% RSLogix 500 project I2P-JOB-15 Duncan_Sutton.RSS, saved by version 10.00.00.00 %
PROJECT "ML01A"    % processor: Bul.1763 MicroLogix 1100 Series B %

PROGRAM FILES
  LAD 2   15 rungs

DATA FILES
  O0 OUTPUT  4 elements
  I1 INPUT  6 elements
  S2 STATUS  66 elements
  B3 BINARY  1 elements
  T4 TIMER  1 elements
  C5 COUNTER  1 elements
  R6 CONTROL  1 elements
  N7 INTEGER  1 elements
  F8 FLOAT  1 elements

LADDER 2
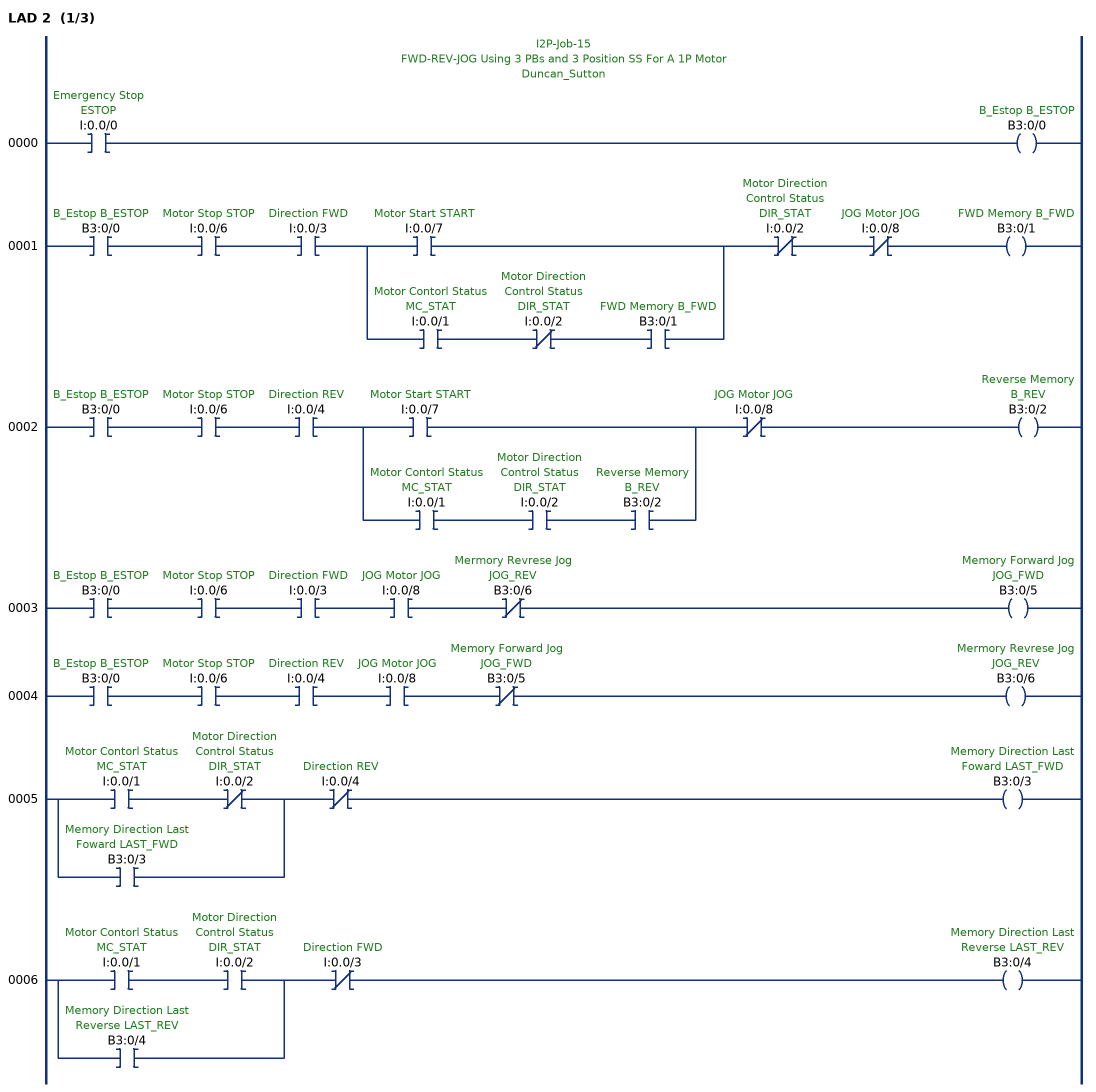
% Rung: 0 %
% I2P-Job-15
% FWD-REV-JOG Using 3 PBs and 3 Position SS For A 1P Motor
% Duncan_Sutton %
SOR XIC I:0.0/0 OTE B3:0/0 EOR
%   I:0.0/0  ESTOP  "Emergency Stop" %
%   B3:0/0  B_ESTOP  "B_Estop" %
% Rung: 1 %
SOR XIC B3:0/0 XIC I:0.0/6 XIC I:0.0/3 BST XIC I:0.0/7 NXB XIC I:0.0/1 XIO I:0.0/2 XIC B3:0/1 BND XIO I:0.0/2 XIO I:0.0/8 OTE B3:0/1 EOR
%   B3:0/0  B_ESTOP  "B_Estop" %
%   I:0.0/6  STOP  "Motor Stop" %
%   I:0.0/3  FWD  "Direction" %
%   I:0.0/7  START  "Motor Start" %
%   I:0.0/1  MC_STAT  "Motor Contorl Status" %
%   I:0.0/2  DIR_STAT  "Motor Direction Control Status" %
%   B3:0/1  B_FWD  "FWD Memory" %
%   I:0.0/8  JOG  "JOG Motor" %
% Rung: 2 %
SOR XIC B3:0/0 XIC I:0.0/6 XIC I:0.0/4 BST XIC I:0.0/7 NXB XIC I:0.0/1 XIC I:0.0/2 XIC B3:0/2 BND XIO I:0.0/8 OTE B3:0/2 EOR
%   B3:0/0  B_ESTOP  "B_Estop" %
%   I:0.0/6  STOP  "Motor Stop" %
%   I:0.0/4  REV  "Direction" %
%   I:0.0/7  START  "Motor Start" %
%   I:0.0/1  MC_STAT  "Motor Contorl Status" %
%   I:0.0/2  DIR_STAT  "Motor Direction Control Status" %
%   B3:0/2  B_REV  "Reverse Memory" %
%   I:0.0/8  JOG  "JOG Motor" %
% Rung: 3 %
SOR XIC B3:0/0 XIC I:0.0/6 XIC I:0.0/3 XIC I:0.0/8 XIO B3:0/6 OTE B3:0/5 EOR
%   B3:0/0  B_ESTOP  "B_Estop" %
%   I:0.0/6  STOP  "Motor Stop" %
%   I:0.0/3  FWD  "Direction" %
%   I:0.0/8  JOG  "JOG Motor" %
%   B3:0/6  JOG_REV  "Mermory Revrese Jog" %
%   B3:0/5  JOG_FWD  "Memory Forward Jog" %
% Rung: 4 %
SOR XIC B3:0/0 XIC I:0.0/6 XIC I:0.0/4 XIC I:0.0/8 XIO B3:0/5 OTE B3:0/6 EOR
%   B3:0/0  B_ESTOP  "B_Estop" %
%   I:0.0/6  STOP  "Motor Stop" %
%   I:0.0/4  REV  "Direction" %
%   I:0.0/8  JOG  "JOG Motor" %
%   B3:0/5  JOG_FWD  "Memory Forward Jog" %
%   B3:0/6  JOG_REV  "Mermory Revrese Jog" %
% Rung: 5 %
SOR BST XIC I:0.0/1 XIO I:0.0/2 NXB XIC B3:0/3 BND XIO I:0.0/4 OTE B3:0/3 EOR
%   I:0.0/1  MC_STAT  "Motor Contorl Status" %
%   I:0.0/2  DIR_STAT  "Motor Direction Control Status" %
%   B3:0/3  LAST_FWD  "Memory Direction Last Foward" %
%   I:0.0/4  REV  "Direction" %
% Rung: 6 %
SOR BST XIC I:0.0/1 XIC I:0.0/2 NXB XIC B3:0/4 BND XIO I:0.0/3 OTE B3:0/4 EOR
%   I:0.0/1  MC_STAT  "Motor Contorl Status" %
%   I:0.0/2  DIR_STAT  "Motor Direction Control Status" %
%   B3:0/4  LAST_REV  "Memory Direction Last Reverse" %
%   I:0.0/3  FWD  "Direction" %

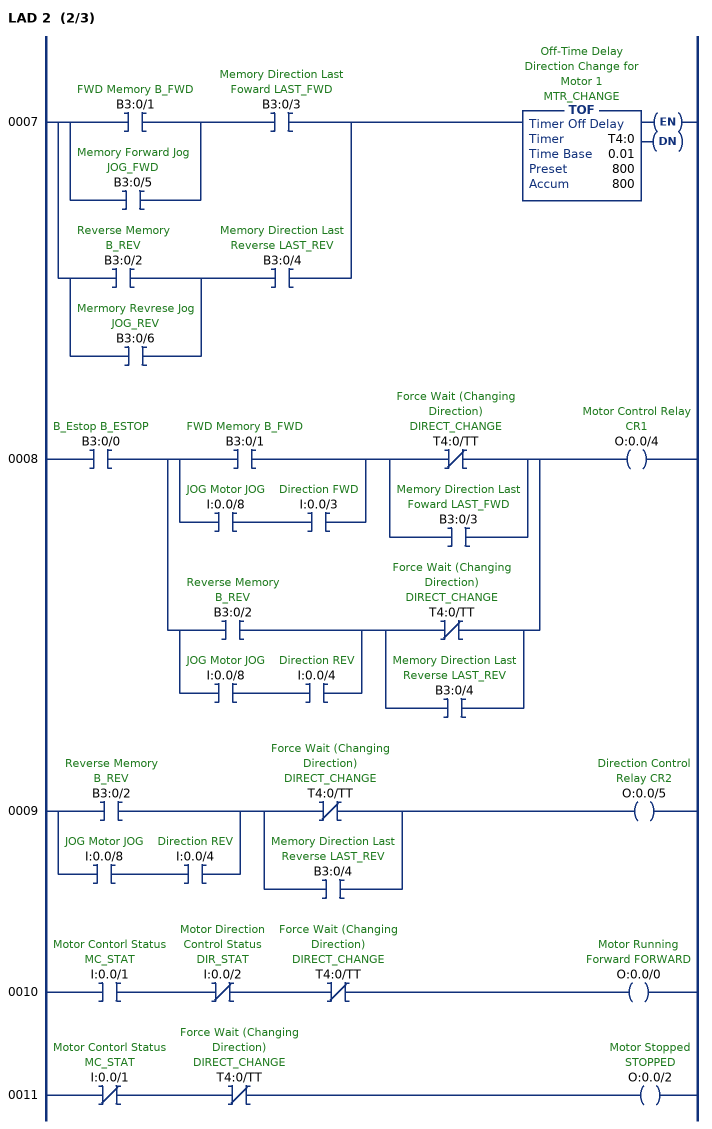
% Rung: 7 %
SOR BST BST XIC B3:0/1 NXB XIC B3:0/5 BND XIC B3:0/3 NXB BST XIC B3:0/2 NXB XIC B3:0/6 BND XIC B3:0/4 BND TOF T4:0 0.01 800 800 EOR
%   B3:0/1  B_FWD  "FWD Memory" %
%   B3:0/5  JOG_FWD  "Memory Forward Jog" %
%   B3:0/3  LAST_FWD  "Memory Direction Last Foward" %
%   B3:0/2  B_REV  "Reverse Memory" %
%   B3:0/6  JOG_REV  "Mermory Revrese Jog" %
%   B3:0/4  LAST_REV  "Memory Direction Last Reverse" %
%   T4:0  MTR_CHANGE  "Off-Time Delay Direction Change for Motor 1" %
% Rung: 8 %
SOR XIC B3:0/0 BST BST XIC B3:0/1 NXB XIC I:0.0/8 XIC I:0.0/3 BND BST XIO T4:0/TT NXB XIC B3:0/3 BND NXB BST XIC B3:0/2 NXB XIC I:0.0/8 XIC I:0.0/4 BND BST XIO T4:0/TT NXB XIC B3:0/4 BND BND OTE O:0.0/4 EOR
%   B3:0/0  B_ESTOP  "B_Estop" %
%   B3:0/1  B_FWD  "FWD Memory" %
%   I:0.0/8  JOG  "JOG Motor" %
%   I:0.0/3  FWD  "Direction" %
%   T4:0/TT  DIRECT_CHANGE  "Force Wait (Changing Direction)" %
%   B3:0/3  LAST_FWD  "Memory Direction Last Foward" %
%   B3:0/2  B_REV  "Reverse Memory" %
%   I:0.0/4  REV  "Direction" %
%   B3:0/4  LAST_REV  "Memory Direction Last Reverse" %
%   O:0.0/4  CR1  "Motor Control Relay" %
% Rung: 9 %
SOR BST XIC B3:0/2 NXB XIC I:0.0/8 XIC I:0.0/4 BND BST XIO T4:0/TT NXB XIC B3:0/4 BND OTE O:0.0/5 EOR
%   B3:0/2  B_REV  "Reverse Memory" %
%   I:0.0/8  JOG  "JOG Motor" %
%   I:0.0/4  REV  "Direction" %
%   T4:0/TT  DIRECT_CHANGE  "Force Wait (Changing Direction)" %
%   B3:0/4  LAST_REV  "Memory Direction Last Reverse" %
%   O:0.0/5  CR2  "Direction Control Relay" %
% Rung: 10 %
SOR XIC I:0.0/1 XIO I:0.0/2 XIO T4:0/TT OTE O:0.0/0 EOR
%   I:0.0/1  MC_STAT  "Motor Contorl Status" %
%   I:0.0/2  DIR_STAT  "Motor Direction Control Status" %
%   T4:0/TT  DIRECT_CHANGE  "Force Wait (Changing Direction)" %
%   O:0.0/0  FORWARD  "Motor Running Forward" %
% Rung: 11 %
SOR XIO I:0.0/1 XIO T4:0/TT OTE O:0.0/2 EOR
%   I:0.0/1  MC_STAT  "Motor Contorl Status" %
%   T4:0/TT  DIRECT_CHANGE  "Force Wait (Changing Direction)" %
%   O:0.0/2  STOPPED  "Motor Stopped" %

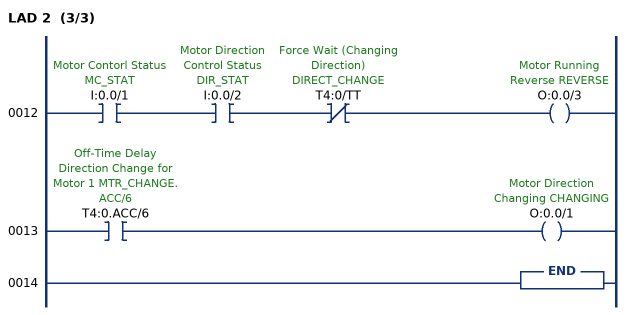
% Rung: 12 %
SOR XIC I:0.0/1 XIC I:0.0/2 XIO T4:0/TT OTE O:0.0/3 EOR
%   I:0.0/1  MC_STAT  "Motor Contorl Status" %
%   I:0.0/2  DIR_STAT  "Motor Direction Control Status" %
%   T4:0/TT  DIRECT_CHANGE  "Force Wait (Changing Direction)" %
%   O:0.0/3  REVERSE  "Motor Running Reverse" %
% Rung: 13 %
SOR XIC T4:0.ACC/6 OTE O:0.0/1 EOR
%   T4:0  MTR_CHANGE  "Off-Time Delay Direction Change for Motor 1" %
%   O:0.0/1  CHANGING  "Motor Direction Changing" %
% Rung: 14 %
SOR END EOR

OTHER DOCUMENTED ADDRESSES
  I:0.0/5  2PSS_PA  "2 Poistion Selector Switch Position A"
  T4:0.ACC/0  T4

DATA TABLE (non-zero values as saved)
DATA B3
% B3:0 % 0X0011
DATA T4
% .PRE .ACC %
% T4:0 % 800 800
